{attribute addProperty BoxType "EP9128-0021-0017"}
{attribute addProperty Id "A_0010_EP9128_0021_0018A_0010_EP9128_0021_0018_B030C9E44664583A_0007_EP9128_0021_0017_2_EP9128_1021EP9128_179A0949162A_0007_EP9128_0021_0017_3_EP9128_2021EP9128_179A0949162"}
{attribute addProperty CRC "1149043925"}
{attribute addProperty SizeInBites "4696"}
{attribute addProperty SizeInBytes "587"}
TYPE A_0007_EP9128_0021_0017_447D04D5 EXTENDS EP9128_179A0949 :
STRUCT
	{attribute addProperty Name "A_0010_EP9128_0021_0018"}
	A_0010_EP9128_0021_0018 : A_0010_EP9128_0021_0018_B030C9E4;
	{attribute addProperty Name "A_0007_EP9128_0021_0017_2_EP9128_1021"}
	A_0007_EP9128_0021_0017_2_EP9128_1021 : EP9128_179A0949;
	{attribute addProperty Name "A_0007_EP9128_0021_0017_3_EP9128_2021"}
	A_0007_EP9128_0021_0017_3_EP9128_2021 : EP9128_179A0949;
END_STRUCT
END_TYPE

(* stored: Version 1.2.0.0, ProductVersion 3.1.4024.9
   DUT A_0007_EP9128_0021_0017_447D04D5: Id {1e058dcd-b4b4-4fcf-a3f8-1216bf1c122c} *)
